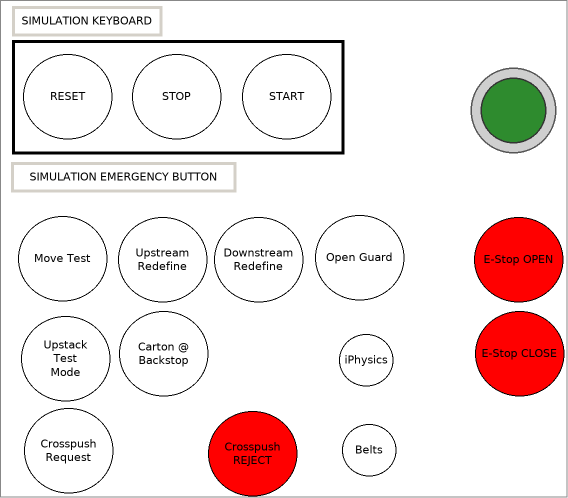
VISUALIZATION Transfer_Keyboard  // 568x498
    Rectangle (12,40 332x114)
    Ellipse (23,54 89x85), "RESET"
        tap csp_transfer_main_services_pushbuttons.visu_reset
    Ellipse (132,54 89x85), "STOP"
        tap csp_transfer_main_services_pushbuttons.visu_stop
    Ellipse (242,54 89x85), "START"
        tap csp_transfer_main_services_pushbuttons.visu_start
    Textfield (12,6 150x30), "SIMULATION KEYBOARD"
    Textfield (11,162 225x30), "SIMULATION EMERGENCY BUTTON"
    Lamp1 (461,61 105x99), variable: csp_transfer_main_safety_emergency.HMI_button_lamp_do.field.status, style: Lamp-Lamp1-Green
    Ellipse (18,216 89x85), "Move Test"
        toggle csp_transfer_upstacker_virtualMaster.move_test_enable
    Ellipse (118,217 89x85), "Upstream Redefine"
        tap csp_transfer_upstacker_virtualMaster.move_test_redefine_upstream
    Ellipse (214,217 89x85), "Downstream Redefine"
        tap csp_transfer_upstacker_virtualMaster.move_test_redefine_downstream
    Ellipse (21,316 89x85), "Upstack Test Mode"
        toggle csp_transfer_upstacker_sensors.debug_active
    Ellipse (119,311 89x85), "Carton @ Backstop"
        toggle csp_transfer_upstacker_sensors.debug_carton_backstop
    Ellipse (24,408 89x85), "Crosspush Request"
        toggle csp_transfer_crosspusher.move_request
    Ellipse (315,215 89x85), "Open Guard"
        toggle csp_transfer_upstacker_virtualMaster.guard_open
    Ellipse (208,411 89x85), "Crosspush REJECT"
        tap csp_transfer_crosspusher_sensors.reject_stack
    Ellipse (339,334 54x52), "iPhysics"
        toggle IP_Main.IP_enable
    Ellipse (474,217 89x85), "E-Stop OPEN"
        tap csp_case_main_services_pushbuttons.visu_emergency_open
    Ellipse (475,311 89x85), "E-Stop CLOSE"
        tap csp_case_main_services_pushbuttons.visu_emergency_close
    Ellipse (342,424 54x52), "Belts"
        toggle csp_transfer_infeed_clamp.start_infeed_belts
END_VISUALIZATION

(* stored: Version 1.1.0.1, ProductVersion 3.1.4024.3
   Visu Transfer_Keyboard: Id {edcf32d1-77ac-4d67-9a47-d75b7cac33e2} *)
